{attribute 'qualified_only'}
VAR_GLOBAL
    timedfb_testshortTime : ULINT;
    timedfb_testLongTime : ULINT;
    statemachinefb_testvariant100 : ULINT;
    statemachinefb_testvariant50 : ULINT;
    statemachinefb_testvariant20 : ULINT;
END_VAR

(* stored: Version 1.1.0.1
   GVL GVL: Id {f215fd48-1cb0-4b73-9578-03c6a30e1dbf} *)
